FUNCTION TryConvert_WORD_TO_USINT : BOOL
VAR_INPUT
	in : WORD;
	out : REFERENCE TO USINT;
END_VAR

IF in > DatatypeLimits.MAX_VALUE_OF_WORD_WHICH_CAN_BE_HELD_IN_A_USINT THEN
	RETURN;
END_IF

out := WORD_TO_USINT(in);
TryConvert_WORD_TO_USINT := TRUE;

END_FUNCTION

(* stored: Version 1.1.0.1, ProductVersion 3.1.4024.12
   POU TryConvert_WORD_TO_USINT: Id {738b9fe4-2c3b-4959-9c63-57ada19e49df}, SpecialFunc None *)
